Yaskawa INFORM job: MAINTENANCE-POSITIO.JBI

/JOB
//NAME MAINTENANCE-POSITIO
//POS
///NPOS 1,0,0,1,0,0
///TOOL 0
///POSTYPE PULSE
///PULSE
C00000=-1,10403,2222,0,7096,0
P00000=0,-222014,-26224,0,-132993,0
//INST
///DATE 2018/08/27 14:52
///ATTR SC,RW
///GROUP1 RB1
NOP
MOVJ P0000 VJ=50.00
MOVL C00000 V=250.0
SETREG MREG#(1) 30
PAUSE
MOVL P0000 V=250.0
END
